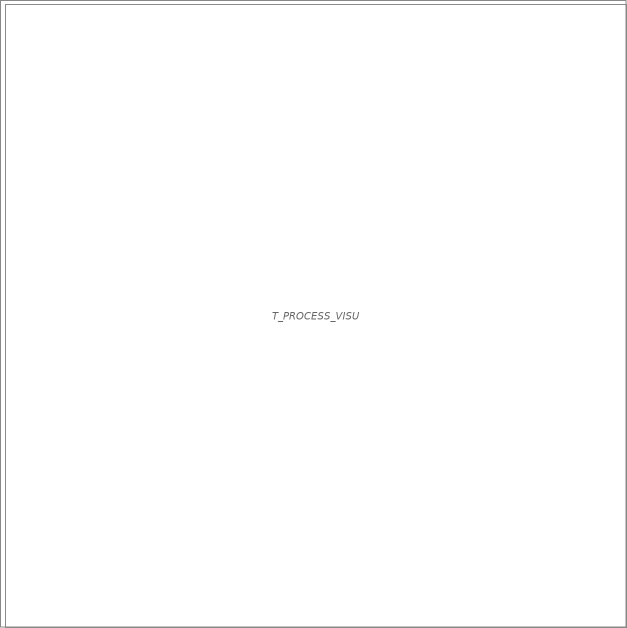
VISUALIZATION PROCESS_CONTROL  // 627x628
    Frame (5,4 622x624)
        shows T_PROCESS_VISU(nSelectedProcess := MAIN.nProcessSelected, EnableProcess := MAIN.wEnableProcess, ProcessCmd := MAIN.eProcessCmd, ProcessState := MAIN.eProcessState, StationState := GVL_XTS.StationState, bStationEnabled := GVL_PROCESS.StationsEnabled)
END_VISUALIZATION

(* stored: Version 1.1.0.1, ProductVersion 3.1.4024.12
   Visu PROCESS_CONTROL: Id {1ba6034d-d395-4dbd-9c83-5ad74be4b21a} *)
